// TIA Portal project "Periyodik Kesme Uygulaması V1" (V16)
// Vorlageprojekt für das Buch mit Zielsystem S7-1200

(* hardware
DEVICE "S7-1200-Station_1"  S7-1200 Station
   slot 0: "Baugruppenträger_0"  Rack  V1.0
   slot 1: "PLC_1"  CPU 1214C DC/DC/DC  6ES7 214-1AG40-0XB0  V4.4
*)

// ===== PLC "PLC_1"  CPU 1214C DC/DC/DC =====

VAR_GLOBAL   // PLC tag table "Standard-Variablentabelle"
   "Sistem_Start_Mem" AT %M10.0 : Bool;
   "Kenar_Darbesi" AT %M10.1 : Bool;
   "Ürün_Sayısı" AT %MW20 : Int;
   "Tag_1" AT %MW30 : Int;
   "Tag_2" AT %MW32 : Int;
   "Tag_3" AT %MW34 : Int;
   "Tag_4" AT %M50.0 : Bool;
   "Tag_5" AT %MW100 : Int;
   "Tag_6" AT %M150.0 : Bool;
   "Tag_7" AT %M150.5 : Bool;
END_VAR

VAR_GLOBAL   // PLC tag table "Tag table_1"
   "Start_But" AT %I0.0 : Bool;
   "Stop_But" AT %I0.1 : Bool;
   "Saati_Setle_But" AT %I0.2 : Bool;
   "Sensör" AT %I0.3 : Bool;
   "Sayıcı_Ekranı" AT %QW30 : Int;
   "Konveyör_1" AT %QW32 : Int;
   "Konveyör_2" AT %QW34 : Int;
   "Konveyör_3" AT %QW36 : Int;
   "Konveyör_4" AT %QW38 : Int;
   "Konveyör_5" AT %QW40 : Int;
END_VAR

DATA_BLOCK "Zaman_Dataları"   // DB1
{ S7_Optimized_Access := 'TRUE' }
VERSION : 0.1
   VAR
      Sistem_Zamanı : DTL;
      Öğle_Zamanı : DTL := DTL#2026-07-24-13:59:00;
      Gece_Çalışması : DTL := DTL#2026-07-24-22:59:00;
   END_VAR
BEGIN
END_DATA_BLOCK

// folder: System blocks/Program resources

DATA_BLOCK "IEC_Counter_0_DB"   // DB2
{ S7_Optimized_Access := 'TRUE' }
AUTHOR : Simatic
FAMILY : IEC
NAME : CNTR
VERSION : 1.0
// stored: InstanceOfName IEC_COUNTER
"IEC_COUNTER"
BEGIN
END_DATA_BLOCK

// folder: (top level)

FUNCTION "MHJ-PLC-Lab-Function-S71200" : Void   // FC9000, SCL
{ S7_Optimized_Access := 'TRUE' }
VERSION : 0.1
   VAR_TEMP
      rdTimeReturn : Int;
      outputTime : DTL;
      SyncVal : Byte;
      forVal : Int;
      forVal_2 : Int;
      Value : Byte;
   END_VAR
   VAR CONSTANT
      CompVal : Byte := 16#34;
      Value_01 : Byte := 16#11;
      Value_01_DW : DWord := 16#A165_D992;
      Value_02_DW : DWord := 16#58BE_4401;
   END_VAR
BEGIN

   #Value:=PEEK(area := 16#82,
        dbNumber := 0,
        byteOffset := 511);
   #Value := #Value + 1;

   POKE(area := 16#82,
        dbNumber := 0,
        byteOffset := 511,
        value := #Value);

   POKE(area:=16#81,
        dbNumber:=0,
        byteOffset:=1016,
        value:=#Value_01_DW);
   POKE(area := 16#81,
        dbNumber := 0,
        byteOffset := 1020,
        value := #Value_02_DW);

   POKE(area := 16#81,
        dbNumber := 0,
        byteOffset := 511,
        value := B#16#00);

   FOR #forVal := 0 TO 120 DO
       FOR #forVal_2:=0 TO 10 DO
           #rdTimeReturn:=RD_SYS_T(#outputTime);
           #rdTimeReturn := WR_SYS_T(#outputTime);
           #rdTimeReturn := RD_SYS_T(#outputTime);
           #rdTimeReturn := WR_SYS_T(#outputTime);
       END_FOR;
       #SyncVal:= PEEK(area := 16#81,
                      dbNumber := 0,
                      byteOffset := 511);
       IF #SyncVal = #CompVal THEN
          GOTO M_1;
       END_IF;
   END_FOR;
   RETURN;

   M_1:
   POKE(area := 16#81,
        dbNumber := 0,
        byteOffset := 511,
        value := B#16#0);
END_FUNCTION

ORGANIZATION_BLOCK "Main"   // OB1, LAD, ProgramCycle
TITLE = "Main Program Sweep (Cycle)"
{ S7_Optimized_Access := 'TRUE' }
VERSION : 0.1
   VAR_INPUT
      Initial_Call : Bool;   // Initial call of this OB
      Remanence : Bool;   // =True, if remanent data are available
   END_VAR
   VAR_TEMP   // added for the SCL form of the ladder/FBD networks
      _w1 : Bool;
      _w2 : Bool;
   END_VAR
BEGIN

REGION Network 1: Connection block for PLCSIM communications. Don't delete this network!
   // Im Netzwerk 1 wird der Konnektierungsbaustein für PLC-Lab aufgerufen.
   // Dieser Aufruf darf nicht entfernt werden!
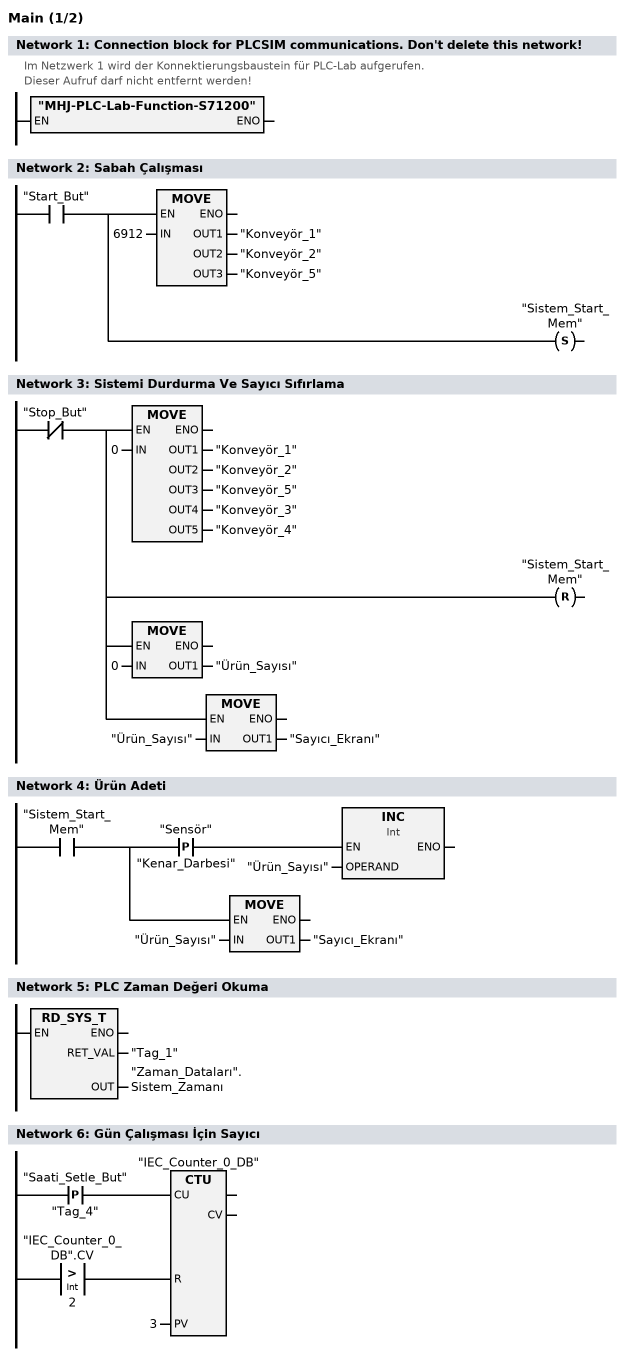
   RUNG wire#powerrail
      "MHJ-PLC-Lab-Function-S71200"()
   END_RUNG
   // the same network as SCL:
   "MHJ-PLC-Lab-Function-S71200"();
END_REGION

REGION Network 2: Sabah Çalışması
   RUNG wire#powerrail
      Contact( "Start_But" )
      wire#w1
      Move(in := 6912, out1 => "Konveyör_1", out2 => "Konveyör_2", out3 => "Konveyör_5")
   END_RUNG
   RUNG wire#w1
      S_Coil( "Sistem_Start_Mem" )
   END_RUNG
   // the same network as SCL:
   IF "Start_But" THEN
       "Konveyör_1" := 6912;
       "Konveyör_2" := 6912;
       "Konveyör_5" := 6912;
       "Sistem_Start_Mem" := TRUE;
   END_IF;
END_REGION

REGION Network 3: Sistemi Durdurma Ve Sayıcı Sıfırlama
   RUNG wire#powerrail
      I_Contact( "Stop_But" )
      wire#w1
      Move(in := 0, out1 => "Konveyör_1", out2 => "Konveyör_2", out3 => "Konveyör_5", out4 => "Konveyör_3", out5 => "Konveyör_4")
   END_RUNG
   RUNG wire#w1
      R_Coil( "Sistem_Start_Mem" )
   END_RUNG
   RUNG wire#w1
      Move(in := 0, out1 => "Ürün_Sayısı")
   END_RUNG
   RUNG wire#w1
      Move(in := "Ürün_Sayısı", out1 => "Sayıcı_Ekranı")
   END_RUNG
   // the same network as SCL:
   IF NOT "Stop_But" THEN
       "Konveyör_1" := 0;
       "Konveyör_2" := 0;
       "Konveyör_5" := 0;
       "Konveyör_3" := 0;
       "Konveyör_4" := 0;
       "Sistem_Start_Mem" := FALSE;
       "Ürün_Sayısı" := 0;
       "Sayıcı_Ekranı" := "Ürün_Sayısı";
   END_IF;
END_REGION

REGION Network 4: Ürün Adeti
   RUNG wire#powerrail
      Contact( "Sistem_Start_Mem" )
      wire#w1
      P_Contact(operand := "Sensör", bit := "Kenar_Darbesi")
      { S7_Templates := "DestType := Int" } Inc( "Ürün_Sayısı" )
   END_RUNG
   RUNG wire#w1
      Move(in := "Ürün_Sayısı", out1 => "Sayıcı_Ekranı")
   END_RUNG
   // the same network as SCL:
   #_w1 := "Sistem_Start_Mem" AND "Sensör" AND NOT "Kenar_Darbesi";   // rising edge of "Sensör"
   "Kenar_Darbesi" := "Sensör";
   IF #_w1 THEN "Ürün_Sayısı" := "Ürün_Sayısı" + 1; END_IF;
   IF "Sistem_Start_Mem" THEN "Sayıcı_Ekranı" := "Ürün_Sayısı"; END_IF;
END_REGION

REGION Network 5: PLC Zaman Değeri Okuma
   "Tag_1" := RD_SYS_T(OUT => "Zaman_Dataları".Sistem_Zamanı);
END_REGION

REGION Network 6: Gün Çalışması İçin Sayıcı
   #_w1 := "Saati_Setle_But" AND NOT "Tag_4";   // rising edge of "Saati_Setle_But"
   "Tag_4" := "Saati_Setle_But";
   "IEC_Counter_0_DB".CTU(CU := #_w1, R := "IEC_Counter_0_DB".CV > 2, PV := 3);
END_REGION

REGION Network 7: Öğlen Çalışması
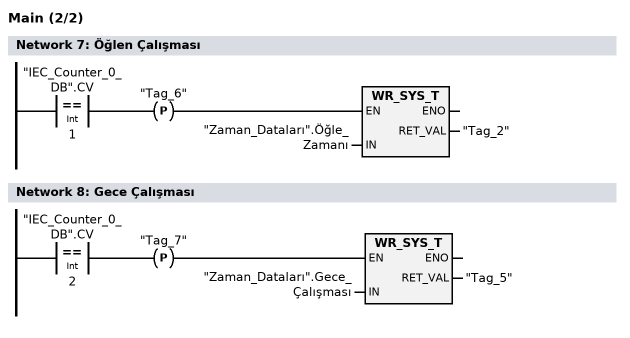
   #_w1 := "IEC_Counter_0_DB".CV = 1;
   #_w2 := #_w1 AND NOT "Tag_6";   // rising edge
   "Tag_6" := #_w1;
   IF #_w2 THEN "Tag_2" := WR_SYS_T(IN := "Zaman_Dataları".Öğle_Zamanı); END_IF;
END_REGION

REGION Network 8: Gece Çalışması
   #_w1 := "IEC_Counter_0_DB".CV = 2;
   #_w2 := #_w1 AND NOT "Tag_7";   // rising edge
   "Tag_7" := #_w1;
   IF #_w2 THEN "Tag_5" := WR_SYS_T(IN := "Zaman_Dataları".Gece_Çalışması); END_IF;
END_REGION
END_ORGANIZATION_BLOCK

ORGANIZATION_BLOCK "Öğlen Çalışması"   // OB10, LAD, TimeOfDay
{ S7_Optimized_Access := 'TRUE' }
VERSION : 0.1
   VAR_INPUT
      CaughtUp : Bool;   // OB call is caught up because time was set forward
      SecondTime : Bool;   // OB call is started a second time because time was set backward
   END_VAR
BEGIN

REGION Network 1: Öğlen Çalışma Programı
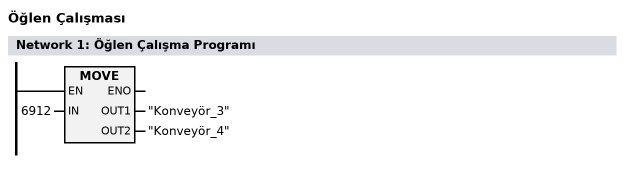
   RUNG wire#powerrail
      Move(in := 6912, out1 => "Konveyör_3", out2 => "Konveyör_4")
   END_RUNG
   // the same network as SCL:
   "Konveyör_3" := 6912;
   "Konveyör_4" := 6912;
END_REGION
END_ORGANIZATION_BLOCK

ORGANIZATION_BLOCK "Gece Çalışması"   // OB11, LAD, TimeOfDay
{ S7_Optimized_Access := 'TRUE' }
VERSION : 0.1
   VAR_INPUT
      CaughtUp : Bool;   // OB call is caught up because time was set forward
      SecondTime : Bool;   // OB call is started a second time because time was set backward
   END_VAR
BEGIN

REGION Network 1: Gece Çalışması
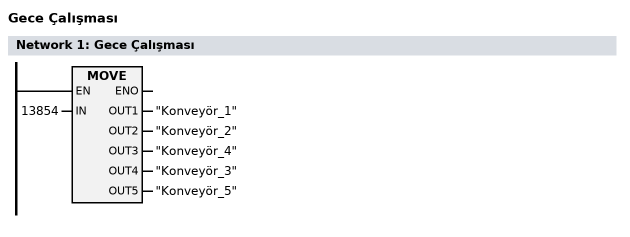
   RUNG wire#powerrail
      Move(in := 13854, out1 => "Konveyör_1", out2 => "Konveyör_2", out3 => "Konveyör_4", out4 => "Konveyör_3", out5 => "Konveyör_5")
   END_RUNG
   // the same network as SCL:
   "Konveyör_1" := 13854;
   "Konveyör_2" := 13854;
   "Konveyör_4" := 13854;
   "Konveyör_3" := 13854;
   "Konveyör_5" := 13854;
END_REGION
END_ORGANIZATION_BLOCK